Staubli VAL3: here.pgx

public program here()
begin
  saveTool:rif2=here(saveTool:gun[0],world)
  saveTool:bCheck=true
end
